FUNCTION F_AbsoluteDecoder : LREAL
VAR_INPUT
		// encoder steps
	input :	ULINT;
	// phase in degrees
	phase : LREAL := 0.0;
	// encoder full turn
	modulus : LREAL := 262144.0;
END_VAR
VAR
	norm : LREAL;
END_VAR

norm := (ULINT_TO_LREAL(input) + modulus - phase*modulus/360.0) / modulus;
F_AbsoluteDecoder := MODABS(norm*360.0, 360.0);

END_FUNCTION

(* stored: Version 1.1.0.1, ProductVersion 3.1.4024.0
   POU F_AbsoluteDecoder: Id {06331f59-fb8f-4087-b1da-febbf7154476}, SpecialFunc None *)
